// TIA Portal V16 export
// export: Created 2024-06-24T15:42:28.6855013Z, ExportSetting WithDefaults, DisplayName Totally Integrated Automation Portal, DisplayVersion V16, DisplayName TIA Portal Version Control Interface, DisplayVersion V16, DisplayName TIA Portal Openness, DisplayVersion V16, DisplayName STEP 7 Professional, DisplayVersion V16, DisplayName STEP 7 Safety, DisplayVersion V16, DisplayName WinCC Advanced, DisplayVersion V16
DATA_BLOCK "DB_Main"   // DB2
VERSION : 0.1
// stored: AutoNumber true, InstanceOfName FB_Main, InstanceOfType FB
"FB_Main"
   // VAR
   //    FB_Conveyor_Entry { S7_SetPoint := 'True'} : "FB_Conveyor";
   //    FB_Conveyor_Weight { S7_SetPoint := 'True'} : "FB_Conveyor";
   //    FB_WheelSorter_Instance { S7_SetPoint := 'True'} : "FB_WheelSorter";
   //    FB_Conveyor_Left { S7_SetPoint := 'True'} : "FB_Conveyor";
   //    FB_Conveyor_Straight { S7_SetPoint := 'True'} : "FB_Conveyor";
   //    FB_Conveyor_Right { S7_SetPoint := 'True'} : "FB_Conveyor";
   //    FB_PickAndPlace_Instance { S7_SetPoint := 'True'} : "FB_PickAndPlace";
   //    FB_Conveyor_4belt { S7_SetPoint := 'True'} : "FB_Conveyor";
   // END_VAR
BEGIN
END_DATA_BLOCK
